{attribute 'qualified_only'}
VAR_GLOBAL
	LogLevel : INT;
END_VAR

(* stored: Version 1.1.0.1
   GVL GVLPluginFramework: Id {1ad4663d-aae7-4491-bdf9-d7f4b936fa2d} *)
